// TIA Portal V20 export
DATA_BLOCK "IDB_HardwareDiag"   // DB12
// stored: InstanceOfName Global.FB_HardwareDiag, InstanceOfType FB, Namespace Global
"Global.FB_HardwareDiag"
   // VAR
   //    ASi { S7_SetPoint := 'True'} : "LineA1.FB_GetDiag";
   // END_VAR
BEGIN
END_DATA_BLOCK
